FUNCTION F_ClearMem : BOOL
VAR_INPUT
    Data : ANY;
END_VAR
VAR
END_VAR

MEMSET(destAddr := Data.pValue,
       fillByte := 0,
       n        := DINT_TO_UDINT(Data.diSize));

END_FUNCTION

(* stored: Version 1.1.0.1, ProductVersion 3.1.4024.12
   POU F_ClearMem: Id {f1b635ea-836d-479e-935f-ca02c0e4e0dd}, SpecialFunc None *)
